TYPE EL5152_CONTROL :
STRUCT

		{attribute 'hide'}
		_reserved1 : BIT;
		{attribute 'hide'}
		_reserved2 : BIT;
		Set_counter : BIT;
		{attribute 'hide'}
		_reserved3 : BIT;
		{attribute 'hide'}
		_reserved4 : BIT;
		{attribute 'hide'}
		_reserved5 : BIT;
		{attribute 'hide'}
		_reserved6 : BIT;
		{attribute 'hide'}
		_reserved7 : BIT;
		{attribute 'hide'}
		_reserved8 : USINT;
		
END_STRUCT
END_TYPE

(* stored: Version 1.1.0.1
   DUT EL5152_CONTROL: Id {b3c70218-a53c-4974-a3c8-126767880847} *)
